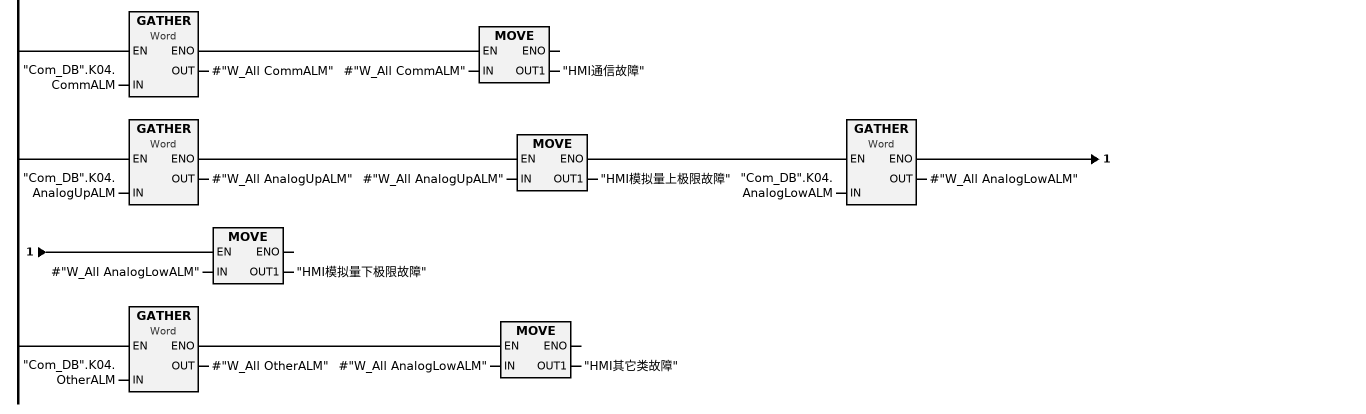
   RUNG wire#powerrail
      { S7_Templates := "[dest_type := Word, src_type := Bool]" } GATHER(IN := "Com_DB".K04.EMO, OUT => #"W_All EMO")
      Move(in := #"W_All EMO", out1 => "HMI总急停报警")
   END_RUNG
   RUNG wire#powerrail
      { S7_Templates := "[dest_type := Word, src_type := Bool]" } GATHER(IN := "Com_DB".K04.SLC, OUT => #"W_All SLC")
      Move(in := #"W_All SLC", out1 => "HMI总光栅报警")
   END_RUNG
   RUNG wire#powerrail
      { S7_Templates := "[dest_type := Word, src_type := Bool]" } GATHER(IN := "Com_DB".K04.DSW, OUT => #"W_All DSW")
      Move(in := #"W_All DSW", out1 => "HMI总安全门报警")
   END_RUNG
   RUNG wire#powerrail
      { S7_Templates := "[dest_type := Word, src_type := Bool]" } GATHER(IN := "Com_DB".K04.OtherSafe, OUT => #"W_All OtherSafe")
      Move(in := #"W_All OtherSafe", out1 => "HMI总其它安全报警")
   END_RUNG
   RUNG wire#powerrail
      { S7_Templates := "[dest_type := Word, src_type := Bool]" } GATHER(IN := "Com_DB".K04.AirALM, OUT => #"W_All AirALM")
      Move(in := #"W_All AirALM", out1 => "HMI总气压报警")
   END_RUNG
   RUNG wire#powerrail
      { S7_Templates := "[dest_type := Word, src_type := Bool, count_type := USInt]" } GATHER_BLK(IN := "Com_DB".K04.SensALM[1], COUNT_OUT := 6, OUT => #"W_All SensALM"[1])
      wire#w1
      Move(in := #"W_All SensALM"[1], out1 => "HMI传感器故障1")
   END_RUNG
   RUNG wire#w1
      Move(in := #"W_All SensALM"[2], out1 => "HMI传感器故障2")
   END_RUNG
   RUNG wire#w1
      Move(in := #"W_All SensALM"[3], out1 => "HMI传感器故障3")
   END_RUNG
   RUNG wire#w1
      Move(in := #"W_All SensALM"[4], out1 => "HMI传感器故障4")
   END_RUNG
   RUNG wire#w1
      Move(in := #"W_All SensALM"[5], out1 => "HMI传感器故障5")
   END_RUNG
   RUNG wire#w1
      Move(in := #"W_All SensALM"[6], out1 => "HMI传感器故障6")
   END_RUNG
   RUNG wire#powerrail
      { S7_Templates := "[dest_type := Word, src_type := Bool, count_type := USInt]" } GATHER_BLK(IN := "Com_DB".K04.MoveALM[1], COUNT_OUT := 3, OUT => #"W_All MoveALM"[1])
      wire#w2
      Move(in := #"W_All MoveALM"[1], out1 => "HMI动作异常1")
   END_RUNG
   RUNG wire#w2
      Move(in := #"W_All MoveALM"[2], out1 => "HMI动作异常2")
   END_RUNG
   RUNG wire#w2
      Move(in := #"W_All MoveALM"[3], out1 => "HMI动作异常3")
   END_RUNG
   RUNG wire#powerrail
      { S7_Templates := "[dest_type := Word, src_type := Bool, count_type := USInt]" } GATHER_BLK(IN := "Com_DB".K04.DrumALM[1], COUNT_OUT := 3, OUT => #"W_All DrumALM"[1])
      wire#w3
      Move(in := #"W_All DrumALM"[1], out1 => "HMI总滚筒故障1")
   END_RUNG
   RUNG wire#w3
      Move(in := #"W_All DrumALM"[2], out1 => "HMI总滚筒故障2")
   END_RUNG
   RUNG wire#w3
      Move(in := #"W_All DrumALM"[1], out1 => "HMI总滚筒故障3")
   END_RUNG
   RUNG wire#powerrail
      { S7_Templates := "[dest_type := Word, src_type := Bool, count_type := USInt]" } GATHER_BLK(IN := "Com_DB".K04.DrumTiOver[1], COUNT_OUT := 3, OUT => #"W_All DrumTiOver"[1])
      wire#w4
      Move(in := #"W_All DrumTiOver"[1], out1 => "HMI总滚筒超时1")
   END_RUNG
   RUNG wire#w4
      Move(in := #"W_All DrumTiOver"[2], out1 => "HMI总滚筒超时2")
   END_RUNG
   RUNG wire#w4
      Move(in := #"W_All DrumTiOver"[3], out1 => "HMI总滚筒超时3")
   END_RUNG
   RUNG wire#powerrail
      { S7_Templates := "[dest_type := Word, src_type := Bool]" } GATHER(IN := "Com_DB".K04.InvALM, OUT => #"W_All InvALM")
      Move(in := #"W_All InvALM", out1 => "HMI总变频器故障")
   END_RUNG
   RUNG wire#powerrail
      { S7_Templates := "[dest_type := Word, src_type := Bool]" } GATHER(IN := "Com_DB".K04.InvNoRun, OUT => #"W_All InvNoRun")
      Move(in := #"W_All InvNoRun", out1 => "HMI总变频器未运行故障")
   END_RUNG
   RUNG wire#powerrail
      { S7_Templates := "[dest_type := Word, src_type := Bool]" } GATHER(IN := "Com_DB".K04.InvOverload, OUT => #"W_All InvOverload")
      Move(in := #"W_All InvOverload", out1 => "HMI总变频器过载故障")
   END_RUNG
   RUNG wire#powerrail
      { S7_Templates := "[dest_type := Word, src_type := Bool]" } GATHER(IN := "Com_DB".K04.InvTiOver, OUT => #"W_All InvTiOver")
      Move(in := #"W_All InvTiOver", out1 => "HMI总变频器超时故障")
   END_RUNG
   RUNG wire#powerrail
      { S7_Templates := "[dest_type := Word, src_type := Bool, count_type := USInt]" } GATHER_BLK(IN := "Com_DB".K04.ValAdvTiOver[1], COUNT_OUT := 3, OUT => #"W_All ValAdvTiOver"[1])
      wire#w5
      { S7_Templates := "[dest_type := Word, src_type := Bool, count_type := USInt]" } GATHER_BLK(IN := "Com_DB".K04.ValRetTiOver[1], COUNT_OUT := 3, OUT => #"W_All ValRetTiOver"[1])
      wire#w6
      Move(in := #"W_All ValRetTiOver"[1], out1 => "HMI阀回动作超时1")
   END_RUNG
   RUNG wire#w6
      Move(in := #"W_All ValRetTiOver"[2], out1 => "HMI阀回动作超时2")
   END_RUNG
   RUNG wire#w6
      Move(in := #"W_All ValRetTiOver"[3], out1 => "HMI阀回动作超时3")
   END_RUNG
   RUNG wire#w5
      Move(in := #"W_All ValAdvTiOver"[1], out1 => "HMI阀出动作超时1")
   END_RUNG
   RUNG wire#w5
      Move(in := #"W_All ValAdvTiOver"[2], out1 => "HMI阀出动作超时2")
   END_RUNG
   RUNG wire#w5
      Move(in := #"W_All ValAdvTiOver"[3], out1 => "HMI阀出动作超时3")
   END_RUNG
   RUNG wire#powerrail
      { S7_Templates := "[dest_type := Word, src_type := Bool, count_type := USInt]" } GATHER_BLK(IN := "Com_DB".K04.ValSensALM[1], COUNT_OUT := 3, OUT => #"W_All ValSensALM"[1])
      wire#w7
      { S7_Templates := "[dest_type := Word, src_type := Bool, count_type := USInt]" } GATHER_BLK(IN := "Com_DB".K04.ValSenCroALM[1], COUNT_OUT := 3, OUT => #"W_All ValSenCroALM"[1])
      wire#w8
      Move(in := #"W_All ValSenCroALM"[1], out1 => "HMI阀传感器交叉ON故障1")
   END_RUNG
   RUNG wire#w8
      Move(in := #"W_All ValSenCroALM"[2], out1 => "HMI阀传感器交叉ON故障2")
   END_RUNG
   RUNG wire#w8
      Move(in := #"W_All ValSenCroALM"[3], out1 => "HMI阀传感器交叉ON故障3")
   END_RUNG
   RUNG wire#w7
      Move(in := #"W_All ValSensALM"[1], out1 => "HMI阀传感器全到位故障1")
   END_RUNG
   RUNG wire#w7
      Move(in := #"W_All ValSensALM"[2], out1 => "HMI阀传感器全到位故障2")
   END_RUNG
   RUNG wire#w7
      Move(in := #"W_All ValSensALM"[3], out1 => "HMI阀传感器全到位故障3")
   END_RUNG
   RUNG wire#powerrail
      { S7_Templates := "[dest_type := Word, src_type := Bool]" } GATHER(IN := "Com_DB".K04.AxisWarn, OUT => #"W_All AxisALM")
      Move(in := #"W_All AxisALM", out1 => "HMI伺服报警")
      { S7_Templates := "[dest_type := Word, src_type := Bool]" } GATHER(IN := "Com_DB".K04.AxisALM, OUT => #"W_All AxisERR")
      Move(in := #"W_All AxisERR", out1 => "HMI伺服故障")
   END_RUNG
   RUNG wire#powerrail
      { S7_Templates := "[dest_type := Word, src_type := Bool]" } GATHER(IN := "Com_DB".K04.AxisNoReady, OUT => #"W_All AxisReady")
      Move(in := #"W_All AxisReady", out1 => "HMI伺服未准备好")
      { S7_Templates := "[dest_type := Word, src_type := Bool]" } GATHER(IN := "Com_DB".K04.AxisHomeALM, OUT => #"W_All AxisHomeALM")
      Move(in := #"W_All AxisHomeALM", out1 => "HMI伺服未回零故障")
   END_RUNG
   RUNG wire#powerrail
      { S7_Templates := "[dest_type := Word, src_type := Bool]" } GATHER(IN := "Com_DB".K04.AxisNoRun, OUT => #"W_All AxisNoRun")
      Move(in := #"W_All AxisNoRun", out1 => "HMI伺服未运行故障")
   END_RUNG
   RUNG wire#powerrail
      { S7_Templates := "[dest_type := Word, src_type := Bool]" } GATHER(IN := "Com_DB".K04.AxisFLS, OUT => #"W_ALL AxisFLSALM")
      Move(in := #"W_ALL AxisFLSALM", out1 => "HM伺服正极限故障")
      { S7_Templates := "[dest_type := Word, src_type := Bool]" } GATHER(IN := "Com_DB".K04.AxisRLS, OUT => #"W_All AxisRLSALM")
      Move(in := #"W_All AxisRLSALM", out1 => "HMI伺服负极限故障")
   END_RUNG
   RUNG wire#powerrail
      { S7_Templates := "[dest_type := Word, src_type := Bool]" } GATHER(IN := "Com_DB".K04.RobotALM, OUT => #"W_All RobotALM")
      Move(in := #"W_All RobotALM", out1 => "HMI机器人故障")
   END_RUNG
   RUNG wire#powerrail
      { S7_Templates := "[dest_type := Word, src_type := Bool]" } GATHER(IN := "Com_DB".K04.CCDALM, OUT => #"W_All CCDALM")
      Move(in := #"W_All CCDALM", out1 => "HMI视觉故障")
   END_RUNG
   RUNG wire#powerrail
      { S7_Templates := "[dest_type := Word, src_type := Bool]" } GATHER(IN := "Com_DB".K04.CommALM, OUT => #"W_All CommALM")
      Move(in := #"W_All CommALM", out1 => "HMI通信故障")
   END_RUNG
   RUNG wire#powerrail
      { S7_Templates := "[dest_type := Word, src_type := Bool]" } GATHER(IN := "Com_DB".K04.AnalogUpALM, OUT => #"W_All AnalogUpALM")
      Move(in := #"W_All AnalogUpALM", out1 => "HMI模拟量上极限故障")
      { S7_Templates := "[dest_type := Word, src_type := Bool]" } GATHER(IN := "Com_DB".K04.AnalogLowALM, OUT => #"W_All AnalogLowALM")
      Move(in := #"W_All AnalogLowALM", out1 => "HMI模拟量下极限故障")
   END_RUNG
   RUNG wire#powerrail
      { S7_Templates := "[dest_type := Word, src_type := Bool]" } GATHER(IN := "Com_DB".K04.OtherALM, OUT => #"W_All OtherALM")
      Move(in := #"W_All AnalogLowALM", out1 => "HMI其它类故障")
   END_RUNG
   // the same network as SCL:
   GATHER(IN := "Com_DB".K04.EMO, OUT => #"W_All EMO", ENO => #_w1);
   IF #_w1 THEN "HMI总急停报警" := #"W_All EMO"; END_IF;
   GATHER(IN := "Com_DB".K04.SLC, OUT => #"W_All SLC", ENO => #_w2);
   IF #_w2 THEN "HMI总光栅报警" := #"W_All SLC"; END_IF;
   GATHER(IN := "Com_DB".K04.DSW, OUT => #"W_All DSW", ENO => #_w3);
   IF #_w3 THEN "HMI总安全门报警" := #"W_All DSW"; END_IF;
   GATHER(IN := "Com_DB".K04.OtherSafe, OUT => #"W_All OtherSafe", ENO => #_w4);
   IF #_w4 THEN "HMI总其它安全报警" := #"W_All OtherSafe"; END_IF;
   GATHER(IN := "Com_DB".K04.AirALM, OUT => #"W_All AirALM", ENO => #_w5);
   IF #_w5 THEN "HMI总气压报警" := #"W_All AirALM"; END_IF;
   GATHER_BLK(IN := "Com_DB".K04.SensALM[1], COUNT_OUT := 6, OUT => #"W_All SensALM"[1], ENO => #_w6);
   IF #_w6 THEN
       "HMI传感器故障1" := #"W_All SensALM"[1];
       "HMI传感器故障2" := #"W_All SensALM"[2];
       "HMI传感器故障3" := #"W_All SensALM"[3];
       "HMI传感器故障4" := #"W_All SensALM"[4];
       "HMI传感器故障5" := #"W_All SensALM"[5];
       "HMI传感器故障6" := #"W_All SensALM"[6];
   END_IF;
   GATHER_BLK(IN := "Com_DB".K04.MoveALM[1], COUNT_OUT := 3, OUT => #"W_All MoveALM"[1], ENO => #_w7);
   IF #_w7 THEN
       "HMI动作异常1" := #"W_All MoveALM"[1];
       "HMI动作异常2" := #"W_All MoveALM"[2];
       "HMI动作异常3" := #"W_All MoveALM"[3];
   END_IF;
   GATHER_BLK(IN := "Com_DB".K04.DrumALM[1], COUNT_OUT := 3, OUT => #"W_All DrumALM"[1], ENO => #_w8);
   IF #_w8 THEN
       "HMI总滚筒故障1" := #"W_All DrumALM"[1];
       "HMI总滚筒故障2" := #"W_All DrumALM"[2];
       "HMI总滚筒故障3" := #"W_All DrumALM"[1];
   END_IF;
   GATHER_BLK(IN := "Com_DB".K04.DrumTiOver[1], COUNT_OUT := 3, OUT => #"W_All DrumTiOver"[1], ENO => #_w9);
   IF #_w9 THEN
       "HMI总滚筒超时1" := #"W_All DrumTiOver"[1];
       "HMI总滚筒超时2" := #"W_All DrumTiOver"[2];
       "HMI总滚筒超时3" := #"W_All DrumTiOver"[3];
   END_IF;
   GATHER(IN := "Com_DB".K04.InvALM, OUT => #"W_All InvALM", ENO => #_w10);
   IF #_w10 THEN "HMI总变频器故障" := #"W_All InvALM"; END_IF;
   GATHER(IN := "Com_DB".K04.InvNoRun, OUT => #"W_All InvNoRun", ENO => #_w11);
   IF #_w11 THEN "HMI总变频器未运行故障" := #"W_All InvNoRun"; END_IF;
   GATHER(IN := "Com_DB".K04.InvOverload, OUT => #"W_All InvOverload", ENO => #_w12);
   IF #_w12 THEN "HMI总变频器过载故障" := #"W_All InvOverload"; END_IF;
   GATHER(IN := "Com_DB".K04.InvTiOver, OUT => #"W_All InvTiOver", ENO => #_w13);
   IF #_w13 THEN "HMI总变频器超时故障" := #"W_All InvTiOver"; END_IF;
   GATHER_BLK(IN := "Com_DB".K04.ValAdvTiOver[1], COUNT_OUT := 3, OUT => #"W_All ValAdvTiOver"[1], ENO => #_w14);
   GATHER_BLK(EN := #_w14,
              IN := "Com_DB".K04.ValRetTiOver[1],
              COUNT_OUT := 3,
              OUT => #"W_All ValRetTiOver"[1],
              ENO => #_w15);
   IF #_w15 THEN
       "HMI阀回动作超时1" := #"W_All ValRetTiOver"[1];
       "HMI阀回动作超时2" := #"W_All ValRetTiOver"[2];
       "HMI阀回动作超时3" := #"W_All ValRetTiOver"[3];
   END_IF;
   IF #_w14 THEN
       "HMI阀出动作超时1" := #"W_All ValAdvTiOver"[1];
       "HMI阀出动作超时2" := #"W_All ValAdvTiOver"[2];
       "HMI阀出动作超时3" := #"W_All ValAdvTiOver"[3];
   END_IF;
   GATHER_BLK(IN := "Com_DB".K04.ValSensALM[1], COUNT_OUT := 3, OUT => #"W_All ValSensALM"[1], ENO => #_w16);
   GATHER_BLK(EN := #_w16,
              IN := "Com_DB".K04.ValSenCroALM[1],
              COUNT_OUT := 3,
              OUT => #"W_All ValSenCroALM"[1],
              ENO => #_w17);
   IF #_w17 THEN
       "HMI阀传感器交叉ON故障1" := #"W_All ValSenCroALM"[1];
       "HMI阀传感器交叉ON故障2" := #"W_All ValSenCroALM"[2];
       "HMI阀传感器交叉ON故障3" := #"W_All ValSenCroALM"[3];
   END_IF;
   IF #_w16 THEN
       "HMI阀传感器全到位故障1" := #"W_All ValSensALM"[1];
       "HMI阀传感器全到位故障2" := #"W_All ValSensALM"[2];
       "HMI阀传感器全到位故障3" := #"W_All ValSensALM"[3];
   END_IF;
   GATHER(IN := "Com_DB".K04.AxisWarn, OUT => #"W_All AxisALM", ENO => #_w18);
   IF #_w18 THEN "HMI伺服报警" := #"W_All AxisALM"; END_IF;
   GATHER(EN := #_w18, IN := "Com_DB".K04.AxisALM, OUT => #"W_All AxisERR", ENO => #_w19);
   IF #_w19 THEN "HMI伺服故障" := #"W_All AxisERR"; END_IF;
   GATHER(IN := "Com_DB".K04.AxisNoReady, OUT => #"W_All AxisReady", ENO => #_w20);
   IF #_w20 THEN "HMI伺服未准备好" := #"W_All AxisReady"; END_IF;
   GATHER(EN := #_w20, IN := "Com_DB".K04.AxisHomeALM, OUT => #"W_All AxisHomeALM", ENO => #_w21);
   IF #_w21 THEN "HMI伺服未回零故障" := #"W_All AxisHomeALM"; END_IF;
   GATHER(IN := "Com_DB".K04.AxisNoRun, OUT => #"W_All AxisNoRun", ENO => #_w22);
   IF #_w22 THEN "HMI伺服未运行故障" := #"W_All AxisNoRun"; END_IF;
   GATHER(IN := "Com_DB".K04.AxisFLS, OUT => #"W_ALL AxisFLSALM", ENO => #_w23);
   IF #_w23 THEN "HM伺服正极限故障" := #"W_ALL AxisFLSALM"; END_IF;
   GATHER(EN := #_w23, IN := "Com_DB".K04.AxisRLS, OUT => #"W_All AxisRLSALM", ENO => #_w24);
   IF #_w24 THEN "HMI伺服负极限故障" := #"W_All AxisRLSALM"; END_IF;
   GATHER(IN := "Com_DB".K04.RobotALM, OUT => #"W_All RobotALM", ENO => #_w25);
   IF #_w25 THEN "HMI机器人故障" := #"W_All RobotALM"; END_IF;
   GATHER(IN := "Com_DB".K04.CCDALM, OUT => #"W_All CCDALM", ENO => #_w26);
   IF #_w26 THEN "HMI视觉故障" := #"W_All CCDALM"; END_IF;
   GATHER(IN := "Com_DB".K04.CommALM, OUT => #"W_All CommALM", ENO => #_w27);
   IF #_w27 THEN "HMI通信故障" := #"W_All CommALM"; END_IF;
   GATHER(IN := "Com_DB".K04.AnalogUpALM, OUT => #"W_All AnalogUpALM", ENO => #_w28);
   IF #_w28 THEN "HMI模拟量上极限故障" := #"W_All AnalogUpALM"; END_IF;
   GATHER(EN := #_w28, IN := "Com_DB".K04.AnalogLowALM, OUT => #"W_All AnalogLowALM", ENO => #_w29);
   IF #_w29 THEN "HMI模拟量下极限故障" := #"W_All AnalogLowALM"; END_IF;
   GATHER(IN := "Com_DB".K04.OtherALM, OUT => #"W_All OtherALM", ENO => #_w30);
   IF #_w30 THEN "HMI其它类故障" := #"W_All AnalogLowALM"; END_IF;
END_REGION

REGION Network 18: 安全类
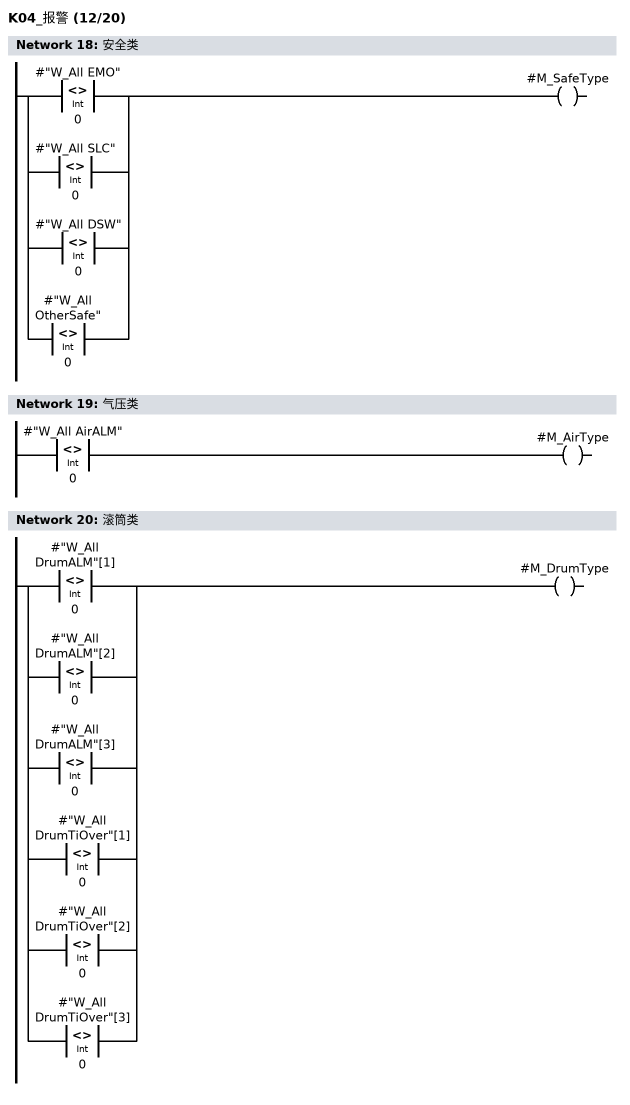
   RUNG wire#powerrail
      { S7_Templates := "SrcType := Int" } NE_Contact(in1 := #"W_All EMO", in2 := 0)
      wire#w1
      Coil( #M_SafeType )
   END_RUNG
   RUNG wire#powerrail
      { S7_Templates := "SrcType := Int" } NE_Contact(in1 := #"W_All SLC", in2 := 0)
   END_RUNG wire#w1
   RUNG wire#powerrail
      { S7_Templates := "SrcType := Int" } NE_Contact(in1 := #"W_All DSW", in2 := 0)
   END_RUNG wire#w1
   RUNG wire#powerrail
      { S7_Templates := "SrcType := Int" } NE_Contact(in1 := #"W_All OtherSafe", in2 := 0)
   END_RUNG wire#w1
   // the same network as SCL:
   #M_SafeType := (#"W_All EMO" <> 0) OR (#"W_All SLC" <> 0) OR (#"W_All DSW" <> 0) OR (#"W_All OtherSafe" <> 0);
END_REGION

REGION Network 19: 气压类
   RUNG wire#powerrail
      { S7_Templates := "SrcType := Int" } NE_Contact(in1 := #"W_All AirALM", in2 := 0)
      Coil( #M_AirType )
   END_RUNG
   // the same network as SCL:
   #M_AirType := #"W_All AirALM" <> 0;
END_REGION

REGION Network 20: 滚筒类
   RUNG wire#powerrail
      { S7_Templates := "SrcType := Int" } NE_Contact(in1 := #"W_All DrumALM"[1], in2 := 0)
      wire#w1
      Coil( #M_DrumType )
   END_RUNG
   RUNG wire#powerrail
      { S7_Templates := "SrcType := Int" } NE_Contact(in1 := #"W_All DrumALM"[2], in2 := 0)
   END_RUNG wire#w1
   RUNG wire#powerrail
      { S7_Templates := "SrcType := Int" } NE_Contact(in1 := #"W_All DrumALM"[3], in2 := 0)
   END_RUNG wire#w1
   RUNG wire#powerrail
      { S7_Templates := "SrcType := Int" } NE_Contact(in1 := #"W_All DrumTiOver"[1], in2 := 0)
   END_RUNG wire#w1
   RUNG wire#powerrail
      { S7_Templates := "SrcType := Int" } NE_Contact(in1 := #"W_All DrumTiOver"[2], in2 := 0)
   END_RUNG wire#w1
   RUNG wire#powerrail
      { S7_Templates := "SrcType := Int" } NE_Contact(in1 := #"W_All DrumTiOver"[3], in2 := 0)
   END_RUNG wire#w1
   // the same network as SCL:
   #M_DrumType := (#"W_All DrumALM"[1] <> 0) OR (#"W_All DrumALM"[2] <> 0) OR (#"W_All DrumALM"[3] <> 0) OR (#"W_All DrumTiOver"[1] <> 0) OR (#"W_All DrumTiOver"[2] <> 0) OR (#"W_All DrumTiOver"[3] <> 0);
END_REGION

REGION Network 21: 变频器类
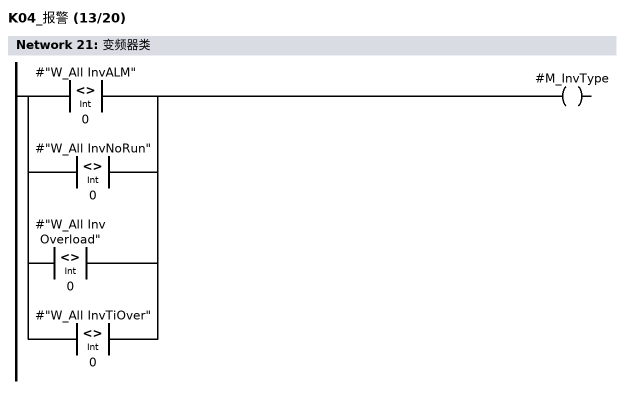
   RUNG wire#powerrail
      { S7_Templates := "SrcType := Int" } NE_Contact(in1 := #"W_All InvALM", in2 := 0)
      wire#w1
      Coil( #M_InvType )
   END_RUNG
   RUNG wire#powerrail
      { S7_Templates := "SrcType := Int" } NE_Contact(in1 := #"W_All InvNoRun", in2 := 0)
   END_RUNG wire#w1
   RUNG wire#powerrail
      { S7_Templates := "SrcType := Int" } NE_Contact(in1 := #"W_All InvOverload", in2 := 0)
   END_RUNG wire#w1
   RUNG wire#powerrail
      { S7_Templates := "SrcType := Int" } NE_Contact(in1 := #"W_All InvTiOver", in2 := 0)
   END_RUNG wire#w1
   // the same network as SCL:
   #M_InvType := (#"W_All InvALM" <> 0) OR (#"W_All InvNoRun" <> 0) OR (#"W_All InvOverload" <> 0) OR (#"W_All InvTiOver" <> 0);
END_REGION

REGION Network 22: 阀类型故障
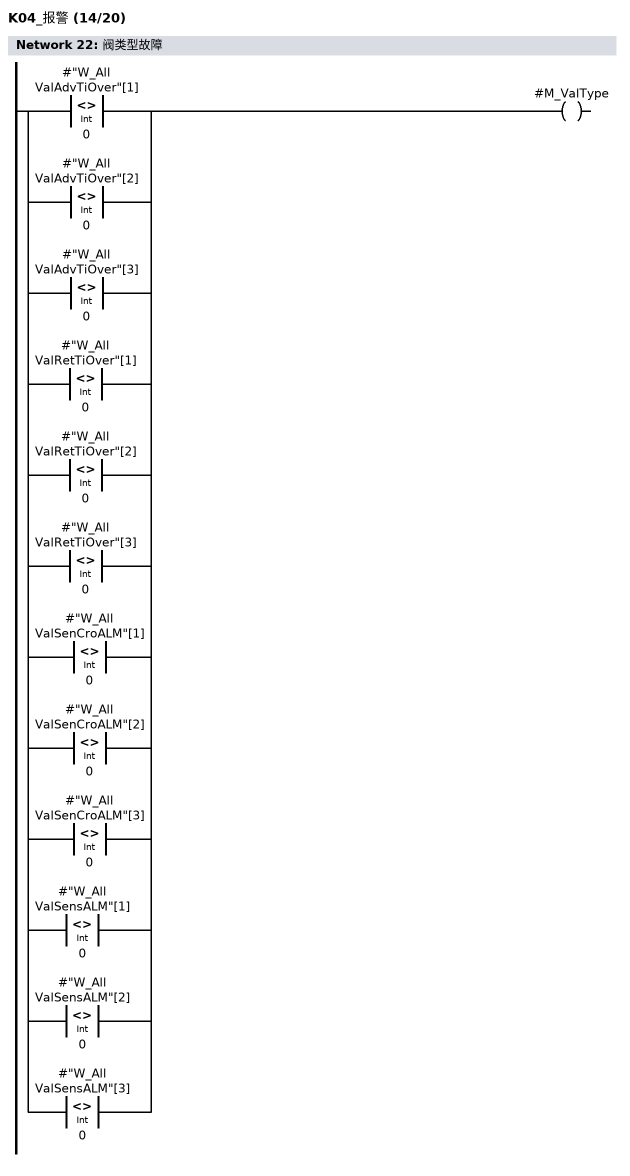
   RUNG wire#powerrail
      { S7_Templates := "SrcType := Int" } NE_Contact(in1 := #"W_All ValAdvTiOver"[1], in2 := 0)
      wire#w1
      Coil( #M_ValType )
   END_RUNG
   RUNG wire#powerrail
      { S7_Templates := "SrcType := Int" } NE_Contact(in1 := #"W_All ValAdvTiOver"[2], in2 := 0)
   END_RUNG wire#w1
   RUNG wire#powerrail
      { S7_Templates := "SrcType := Int" } NE_Contact(in1 := #"W_All ValAdvTiOver"[3], in2 := 0)
   END_RUNG wire#w1
   RUNG wire#powerrail
      { S7_Templates := "SrcType := Int" } NE_Contact(in1 := #"W_All ValRetTiOver"[1], in2 := 0)
   END_RUNG wire#w1
   RUNG wire#powerrail
      { S7_Templates := "SrcType := Int" } NE_Contact(in1 := #"W_All ValRetTiOver"[2], in2 := 0)
   END_RUNG wire#w1
   RUNG wire#powerrail
      { S7_Templates := "SrcType := Int" } NE_Contact(in1 := #"W_All ValRetTiOver"[3], in2 := 0)
   END_RUNG wire#w1
   RUNG wire#powerrail
      { S7_Templates := "SrcType := Int" } NE_Contact(in1 := #"W_All ValSenCroALM"[1], in2 := 0)
   END_RUNG wire#w1
   RUNG wire#powerrail
      { S7_Templates := "SrcType := Int" } NE_Contact(in1 := #"W_All ValSenCroALM"[2], in2 := 0)
   END_RUNG wire#w1
   RUNG wire#powerrail
      { S7_Templates := "SrcType := Int" } NE_Contact(in1 := #"W_All ValSenCroALM"[3], in2 := 0)
   END_RUNG wire#w1
   RUNG wire#powerrail
      { S7_Templates := "SrcType := Int" } NE_Contact(in1 := #"W_All ValSensALM"[1], in2 := 0)
   END_RUNG wire#w1
   RUNG wire#powerrail
      { S7_Templates := "SrcType := Int" } NE_Contact(in1 := #"W_All ValSensALM"[2], in2 := 0)
   END_RUNG wire#w1
   RUNG wire#powerrail
      { S7_Templates := "SrcType := Int" } NE_Contact(in1 := #"W_All ValSensALM"[3], in2 := 0)
   END_RUNG wire#w1
   // the same network as SCL:
   #M_ValType := (#"W_All ValAdvTiOver"[1] <> 0) OR (#"W_All ValAdvTiOver"[2] <> 0) OR (#"W_All ValAdvTiOver"[3] <> 0) OR (#"W_All ValRetTiOver"[1] <> 0) OR (#"W_All ValRetTiOver"[2] <> 0) OR (#"W_All ValRetTiOver"[3] <> 0) OR (#"W_All ValSenCroALM"[1] <> 0) OR (#"W_All ValSenCroALM"[2] <> 0) OR (#"W_All ValSenCroALM"[3] <> 0) OR (#"W_All ValSensALM"[1] <> 0) OR (#"W_All ValSensALM"[2] <> 0) OR (#"W_All ValSensALM"[3] <> 0);
END_REGION

REGION Network 23: 伺服类别
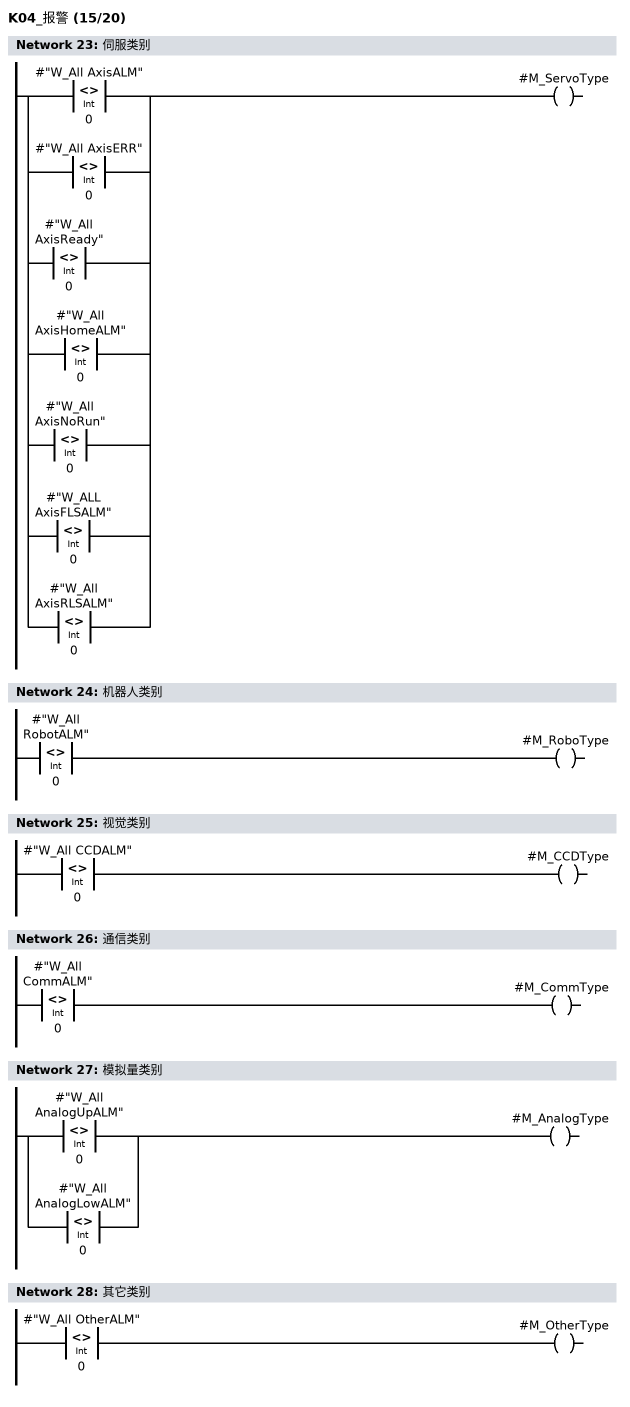
   RUNG wire#powerrail
      { S7_Templates := "SrcType := Int" } NE_Contact(in1 := #"W_All AxisALM", in2 := 0)
      wire#w1
      Coil( #M_ServoType )
   END_RUNG
   RUNG wire#powerrail
      { S7_Templates := "SrcType := Int" } NE_Contact(in1 := #"W_All AxisERR", in2 := 0)
   END_RUNG wire#w1
   RUNG wire#powerrail
      { S7_Templates := "SrcType := Int" } NE_Contact(in1 := #"W_All AxisReady", in2 := 0)
   END_RUNG wire#w1
   RUNG wire#powerrail
      { S7_Templates := "SrcType := Int" } NE_Contact(in1 := #"W_All AxisHomeALM", in2 := 0)
   END_RUNG wire#w1
   RUNG wire#powerrail
      { S7_Templates := "SrcType := Int" } NE_Contact(in1 := #"W_All AxisNoRun", in2 := 0)
   END_RUNG wire#w1
   RUNG wire#powerrail
      { S7_Templates := "SrcType := Int" } NE_Contact(in1 := #"W_ALL AxisFLSALM", in2 := 0)
   END_RUNG wire#w1
   RUNG wire#powerrail
      { S7_Templates := "SrcType := Int" } NE_Contact(in1 := #"W_All AxisRLSALM", in2 := 0)
   END_RUNG wire#w1
   // the same network as SCL:
   #M_ServoType := (#"W_All AxisALM" <> 0) OR (#"W_All AxisERR" <> 0) OR (#"W_All AxisReady" <> 0) OR (#"W_All AxisHomeALM" <> 0) OR (#"W_All AxisNoRun" <> 0) OR (#"W_ALL AxisFLSALM" <> 0) OR (#"W_All AxisRLSALM" <> 0);
END_REGION

REGION Network 24: 机器人类别
   RUNG wire#powerrail
      { S7_Templates := "SrcType := Int" } NE_Contact(in1 := #"W_All RobotALM", in2 := 0)
      Coil( #M_RoboType )
   END_RUNG
   // the same network as SCL:
   #M_RoboType := #"W_All RobotALM" <> 0;
END_REGION

REGION Network 25: 视觉类别
   RUNG wire#powerrail
      { S7_Templates := "SrcType := Int" } NE_Contact(in1 := #"W_All CCDALM", in2 := 0)
      Coil( #M_CCDType )
   END_RUNG
   // the same network as SCL:
   #M_CCDType := #"W_All CCDALM" <> 0;
END_REGION

REGION Network 26: 通信类别
   RUNG wire#powerrail
      { S7_Templates := "SrcType := Int" } NE_Contact(in1 := #"W_All CommALM", in2 := 0)
      Coil( #M_CommType )
   END_RUNG
   // the same network as SCL:
   #M_CommType := #"W_All CommALM" <> 0;
END_REGION

REGION Network 27: 模拟量类别
   RUNG wire#powerrail
      { S7_Templates := "SrcType := Int" } NE_Contact(in1 := #"W_All AnalogUpALM", in2 := 0)
      wire#w1
      Coil( #M_AnalogType )
   END_RUNG
   RUNG wire#powerrail
      { S7_Templates := "SrcType := Int" } NE_Contact(in1 := #"W_All AnalogLowALM", in2 := 0)
   END_RUNG wire#w1
   // the same network as SCL:
   #M_AnalogType := (#"W_All AnalogUpALM" <> 0) OR (#"W_All AnalogLowALM" <> 0);
END_REGION

REGION Network 28: 其它类别
   RUNG wire#powerrail
      { S7_Templates := "SrcType := Int" } NE_Contact(in1 := #"W_All OtherALM", in2 := 0)
      Coil( #M_OtherType )
   END_RUNG
   // the same network as SCL:
   #M_OtherType := #"W_All OtherALM" <> 0;
END_REGION

REGION Network 29: 传感器故障类
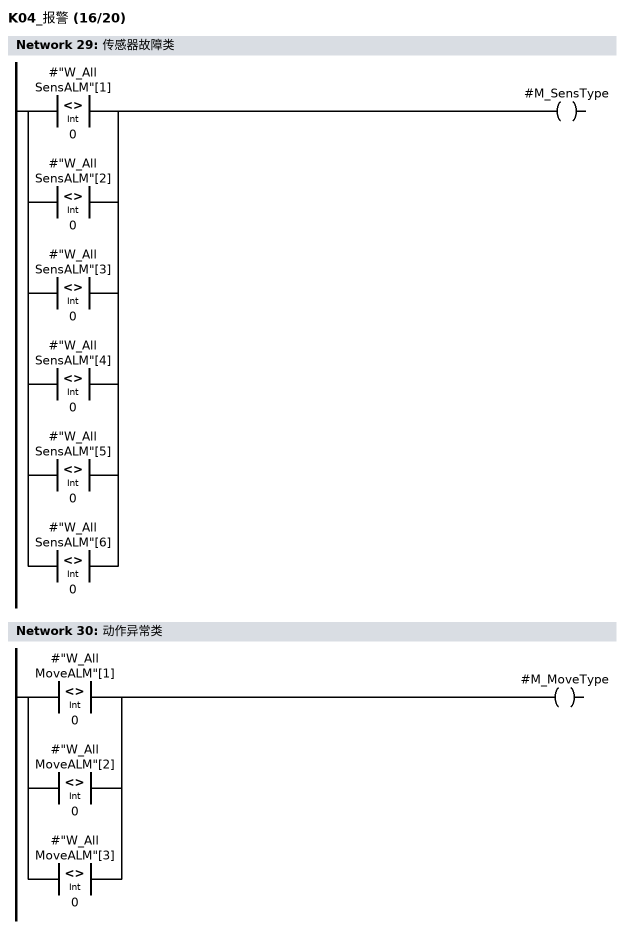
   RUNG wire#powerrail
      { S7_Templates := "SrcType := Int" } NE_Contact(in1 := #"W_All SensALM"[1], in2 := 0)
      wire#w1
      Coil( #M_SensType )
   END_RUNG
   RUNG wire#powerrail
      { S7_Templates := "SrcType := Int" } NE_Contact(in1 := #"W_All SensALM"[2], in2 := 0)
   END_RUNG wire#w1
   RUNG wire#powerrail
      { S7_Templates := "SrcType := Int" } NE_Contact(in1 := #"W_All SensALM"[3], in2 := 0)
   END_RUNG wire#w1
   RUNG wire#powerrail
      { S7_Templates := "SrcType := Int" } NE_Contact(in1 := #"W_All SensALM"[4], in2 := 0)
   END_RUNG wire#w1
   RUNG wire#powerrail
      { S7_Templates := "SrcType := Int" } NE_Contact(in1 := #"W_All SensALM"[5], in2 := 0)
   END_RUNG wire#w1
   RUNG wire#powerrail
      { S7_Templates := "SrcType := Int" } NE_Contact(in1 := #"W_All SensALM"[6], in2 := 0)
   END_RUNG wire#w1
   // the same network as SCL:
   #M_SensType := (#"W_All SensALM"[1] <> 0) OR (#"W_All SensALM"[2] <> 0) OR (#"W_All SensALM"[3] <> 0) OR (#"W_All SensALM"[4] <> 0) OR (#"W_All SensALM"[5] <> 0) OR (#"W_All SensALM"[6] <> 0);
END_REGION

REGION Network 30: 动作异常类
   RUNG wire#powerrail
      { S7_Templates := "SrcType := Int" } NE_Contact(in1 := #"W_All MoveALM"[1], in2 := 0)
      wire#w1
      Coil( #M_MoveType )
   END_RUNG
   RUNG wire#powerrail
      { S7_Templates := "SrcType := Int" } NE_Contact(in1 := #"W_All MoveALM"[2], in2 := 0)
   END_RUNG wire#w1
   RUNG wire#powerrail
      { S7_Templates := "SrcType := Int" } NE_Contact(in1 := #"W_All MoveALM"[3], in2 := 0)
   END_RUNG wire#w1
   // the same network as SCL:
   #M_MoveType := (#"W_All MoveALM"[1] <> 0) OR (#"W_All MoveALM"[2] <> 0) OR (#"W_All MoveALM"[3] <> 0);
END_REGION

REGION Network 31: 故障汇总
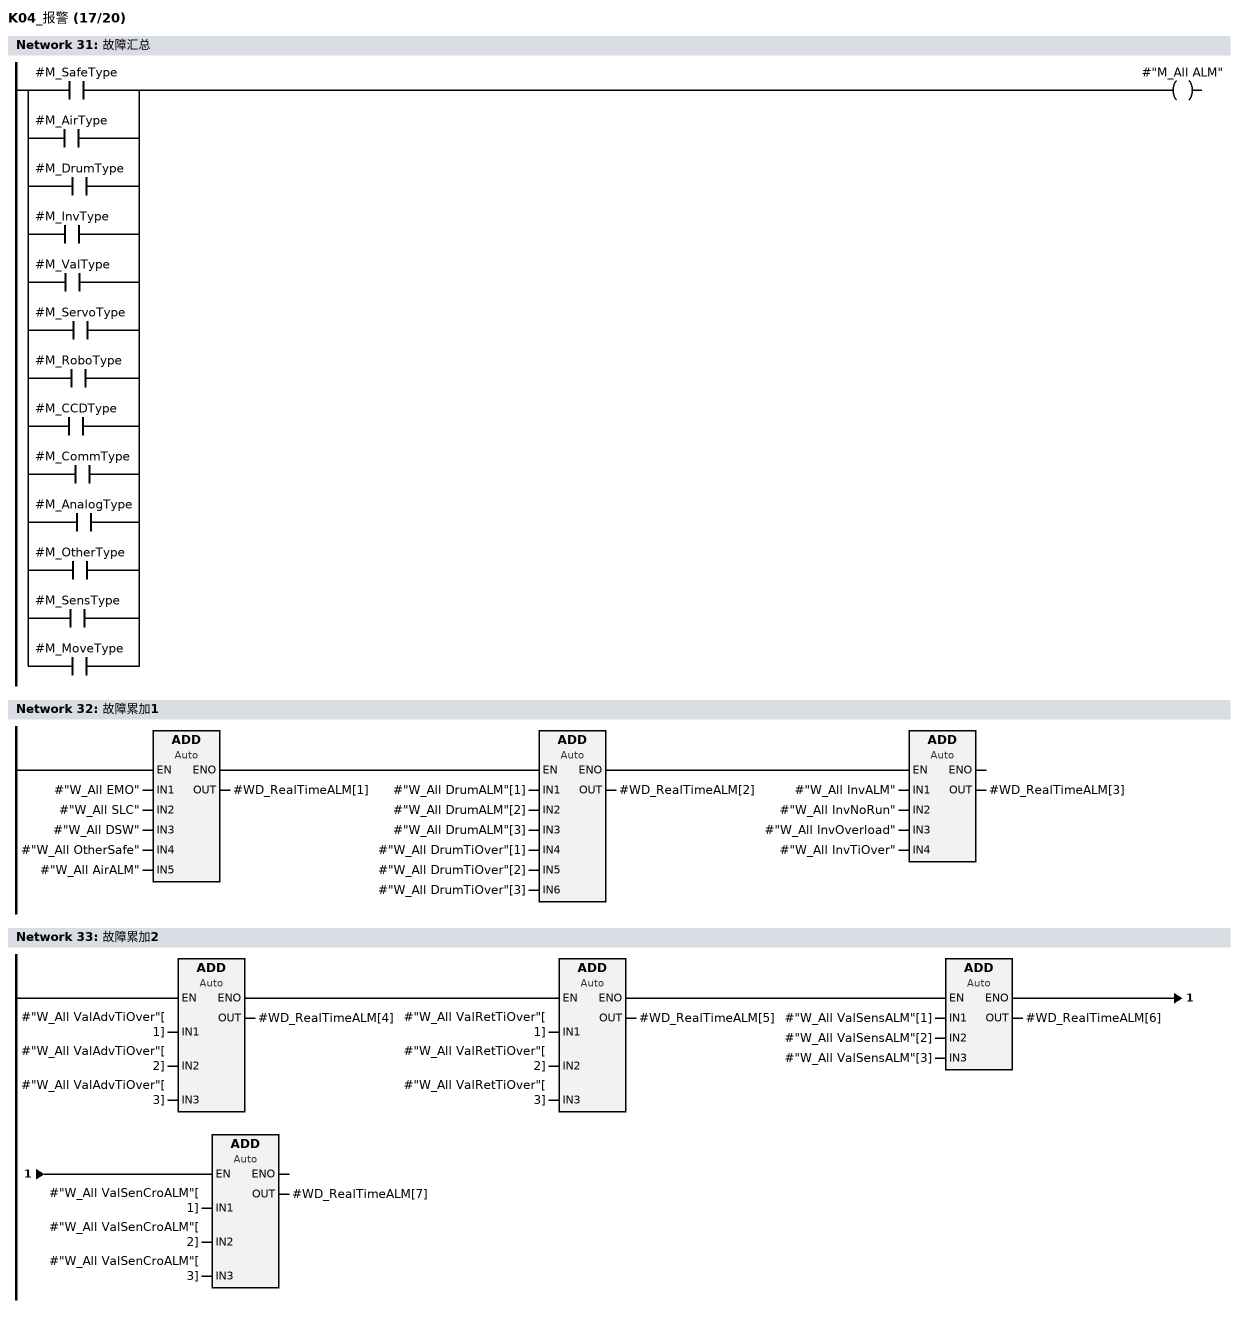
   RUNG wire#powerrail
      Contact( #M_SafeType )
      wire#w1
      Coil( #"M_All ALM" )
   END_RUNG
   RUNG wire#powerrail
      Contact( #M_AirType )
   END_RUNG wire#w1
   RUNG wire#powerrail
      Contact( #M_DrumType )
   END_RUNG wire#w1
   RUNG wire#powerrail
      Contact( #M_InvType )
   END_RUNG wire#w1
   RUNG wire#powerrail
      Contact( #M_ValType )
   END_RUNG wire#w1
   RUNG wire#powerrail
      Contact( #M_ServoType )
   END_RUNG wire#w1
   RUNG wire#powerrail
      Contact( #M_RoboType )
   END_RUNG wire#w1
   RUNG wire#powerrail
      Contact( #M_CCDType )
   END_RUNG wire#w1
   RUNG wire#powerrail
      Contact( #M_CommType )
   END_RUNG wire#w1
   RUNG wire#powerrail
      Contact( #M_AnalogType )
   END_RUNG wire#w1
   RUNG wire#powerrail
      Contact( #M_OtherType )
   END_RUNG wire#w1
   RUNG wire#powerrail
      Contact( #M_SensType )
   END_RUNG wire#w1
   RUNG wire#powerrail
      Contact( #M_MoveType )
   END_RUNG wire#w1
   // the same network as SCL:
   #"M_All ALM" := #M_SafeType OR #M_AirType OR #M_DrumType OR #M_InvType OR #M_ValType OR #M_ServoType OR #M_RoboType OR #M_CCDType OR #M_CommType OR #M_AnalogType OR #M_OtherType OR #M_SensType OR #M_MoveType;
END_REGION

REGION Network 32: 故障累加1
   RUNG wire#powerrail
      Add(in1 := #"W_All EMO", in2 := #"W_All SLC", in3 := #"W_All DSW", in4 := #"W_All OtherSafe", in5 := #"W_All AirALM", out => #WD_RealTimeALM[1])
      Add(in1 := #"W_All DrumALM"[1], in2 := #"W_All DrumALM"[2], in3 := #"W_All DrumALM"[3], in4 := #"W_All DrumTiOver"[1], in5 := #"W_All DrumTiOver"[2], in6 := #"W_All DrumTiOver"[3], out => #WD_RealTimeALM[2])
      Add(in1 := #"W_All InvALM", in2 := #"W_All InvNoRun", in3 := #"W_All InvOverload", in4 := #"W_All InvTiOver", out => #WD_RealTimeALM[3])
   END_RUNG
   // the same network as SCL:
   #WD_RealTimeALM[1] := #"W_All EMO" + #"W_All SLC" + #"W_All DSW" + #"W_All OtherSafe" + #"W_All AirALM";
   #WD_RealTimeALM[2] := #"W_All DrumALM"[1] + #"W_All DrumALM"[2] + #"W_All DrumALM"[3] + #"W_All DrumTiOver"[1] + #"W_All DrumTiOver"[2] + #"W_All DrumTiOver"[3];
   #WD_RealTimeALM[3] := #"W_All InvALM" + #"W_All InvNoRun" + #"W_All InvOverload" + #"W_All InvTiOver";
END_REGION

REGION Network 33: 故障累加2
   RUNG wire#powerrail
      Add(in1 := #"W_All ValAdvTiOver"[1], in2 := #"W_All ValAdvTiOver"[2], in3 := #"W_All ValAdvTiOver"[3], out => #WD_RealTimeALM[4])
      Add(in1 := #"W_All ValRetTiOver"[1], in2 := #"W_All ValRetTiOver"[2], in3 := #"W_All ValRetTiOver"[3], out => #WD_RealTimeALM[5])
      Add(in1 := #"W_All ValSensALM"[1], in2 := #"W_All ValSensALM"[2], in3 := #"W_All ValSensALM"[3], out => #WD_RealTimeALM[6])
      Add(in1 := #"W_All ValSenCroALM"[1], in2 := #"W_All ValSenCroALM"[2], in3 := #"W_All ValSenCroALM"[3], out => #WD_RealTimeALM[7])
   END_RUNG
   // the same network as SCL:
   #WD_RealTimeALM[4] := #"W_All ValAdvTiOver"[1] + #"W_All ValAdvTiOver"[2] + #"W_All ValAdvTiOver"[3];
   #WD_RealTimeALM[5] := #"W_All ValRetTiOver"[1] + #"W_All ValRetTiOver"[2] + #"W_All ValRetTiOver"[3];
   #WD_RealTimeALM[6] := #"W_All ValSensALM"[1] + #"W_All ValSensALM"[2] + #"W_All ValSensALM"[3];
   #WD_RealTimeALM[7] := #"W_All ValSenCroALM"[1] + #"W_All ValSenCroALM"[2] + #"W_All ValSenCroALM"[3];
END_REGION

REGION Network 34: 故障累加3
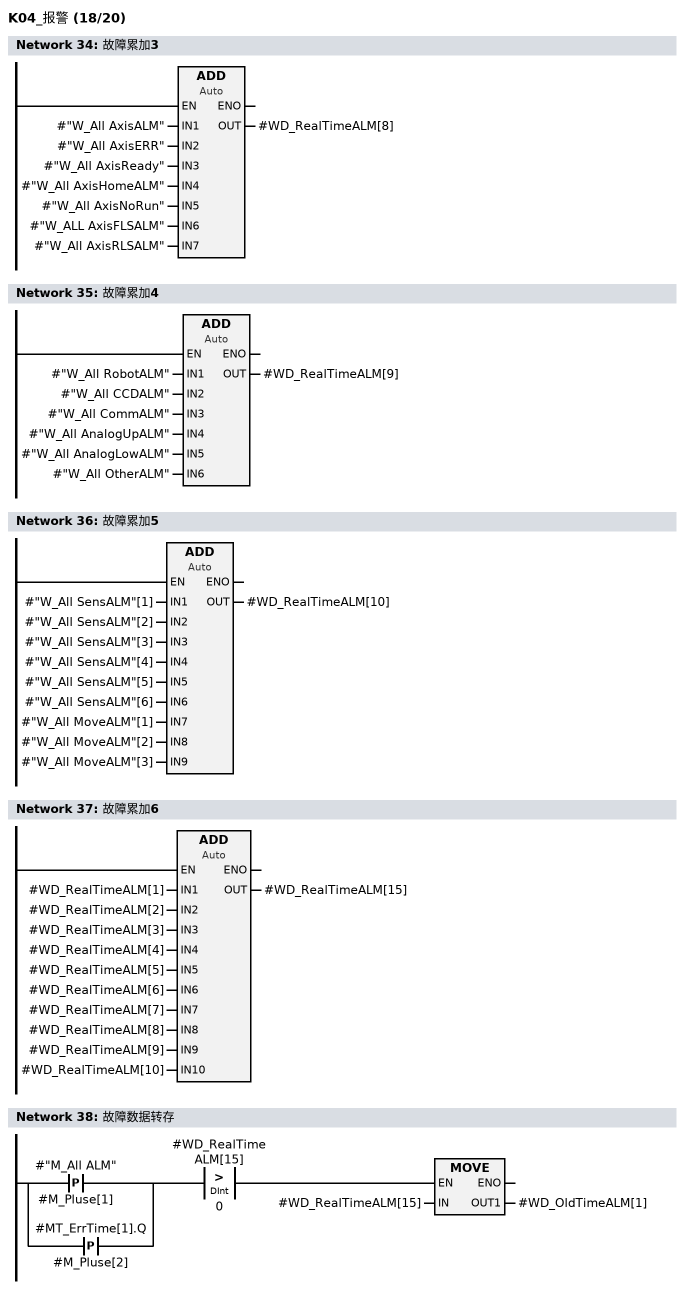
   RUNG wire#powerrail
      Add(in1 := #"W_All AxisALM", in2 := #"W_All AxisERR", in3 := #"W_All AxisReady", in4 := #"W_All AxisHomeALM", in5 := #"W_All AxisNoRun", in6 := #"W_ALL AxisFLSALM", in7 := #"W_All AxisRLSALM", out => #WD_RealTimeALM[8])
   END_RUNG
   // the same network as SCL:
   #WD_RealTimeALM[8] := #"W_All AxisALM" + #"W_All AxisERR" + #"W_All AxisReady" + #"W_All AxisHomeALM" + #"W_All AxisNoRun" + #"W_ALL AxisFLSALM" + #"W_All AxisRLSALM";
END_REGION

REGION Network 35: 故障累加4
   RUNG wire#powerrail
      Add(in1 := #"W_All RobotALM", in2 := #"W_All CCDALM", in3 := #"W_All CommALM", in4 := #"W_All AnalogUpALM", in5 := #"W_All AnalogLowALM", in6 := #"W_All OtherALM", out => #WD_RealTimeALM[9])
   END_RUNG
   // the same network as SCL:
   #WD_RealTimeALM[9] := #"W_All RobotALM" + #"W_All CCDALM" + #"W_All CommALM" + #"W_All AnalogUpALM" + #"W_All AnalogLowALM" + #"W_All OtherALM";
END_REGION

REGION Network 36: 故障累加5
   RUNG wire#powerrail
      Add(in1 := #"W_All SensALM"[1], in2 := #"W_All SensALM"[2], in3 := #"W_All SensALM"[3], in4 := #"W_All SensALM"[4], in5 := #"W_All SensALM"[5], in6 := #"W_All SensALM"[6], in7 := #"W_All MoveALM"[1], in8 := #"W_All MoveALM"[2], in9 := #"W_All MoveALM"[3], out => #WD_RealTimeALM[10])
   END_RUNG
   // the same network as SCL:
   #WD_RealTimeALM[10] := #"W_All SensALM"[1] + #"W_All SensALM"[2] + #"W_All SensALM"[3] + #"W_All SensALM"[4] + #"W_All SensALM"[5] + #"W_All SensALM"[6] + #"W_All MoveALM"[1] + #"W_All MoveALM"[2] + #"W_All MoveALM"[3];
END_REGION

REGION Network 37: 故障累加6
   RUNG wire#powerrail
      Add(in1 := #WD_RealTimeALM[1], in2 := #WD_RealTimeALM[2], in3 := #WD_RealTimeALM[3], in4 := #WD_RealTimeALM[4], in5 := #WD_RealTimeALM[5], in6 := #WD_RealTimeALM[6], in7 := #WD_RealTimeALM[7], in8 := #WD_RealTimeALM[8], in9 := #WD_RealTimeALM[9], in10 := #WD_RealTimeALM[10], out => #WD_RealTimeALM[15])
   END_RUNG
   // the same network as SCL:
   #WD_RealTimeALM[15] := #WD_RealTimeALM[1] + #WD_RealTimeALM[2] + #WD_RealTimeALM[3] + #WD_RealTimeALM[4] + #WD_RealTimeALM[5] + #WD_RealTimeALM[6] + #WD_RealTimeALM[7] + #WD_RealTimeALM[8] + #WD_RealTimeALM[9] + #WD_RealTimeALM[10];
END_REGION

REGION Network 38: 故障数据转存
   RUNG wire#powerrail
      P_Contact(operand := #"M_All ALM", bit := #M_Pluse[1])
      wire#w1
      { S7_Templates := "SrcType := DInt" } GT_Contact(in1 := #WD_RealTimeALM[15], in2 := 0)
      Move(in := #WD_RealTimeALM[15], out1 => #WD_OldTimeALM[1])
   END_RUNG
   RUNG wire#powerrail
      P_Contact(operand := #MT_ErrTime[1].Q, bit := #M_Pluse[2])
   END_RUNG wire#w1
   // the same network as SCL:
   #_w1 := #"M_All ALM" AND NOT #M_Pluse[1];   // rising edge of #"M_All ALM"
   #M_Pluse[1] := #"M_All ALM";
   #_w2 := #MT_ErrTime[1].Q AND NOT #M_Pluse[2];   // rising edge of #MT_ErrTime[1].Q
   #M_Pluse[2] := #MT_ErrTime[1].Q;
   IF (#_w1 OR #_w2) AND (#WD_RealTimeALM[15] > 0) THEN #WD_OldTimeALM[1] := #WD_RealTimeALM[15]; END_IF;
END_REGION

REGION Network 39: 故障汇总新的
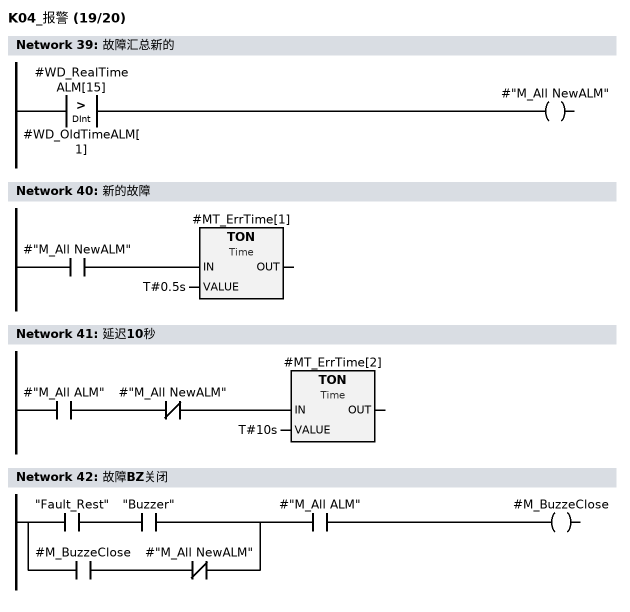
   RUNG wire#powerrail
      { S7_Templates := "SrcType := DInt" } GT_Contact(in1 := #WD_RealTimeALM[15], in2 := #WD_OldTimeALM[1])
      Coil( #"M_All NewALM" )
   END_RUNG
   // the same network as SCL:
   #"M_All NewALM" := #WD_RealTimeALM[15] > #WD_OldTimeALM[1];
END_REGION

REGION Network 40: 新的故障
   #MT_ErrTime[1].TON(IN := #"M_All NewALM", PT := T#0.5s);   // TON coil
END_REGION

REGION Network 41: 延迟10秒
   #MT_ErrTime[2].TON(IN := #"M_All ALM" AND NOT #"M_All NewALM", PT := T#10s);   // TON coil
END_REGION

REGION Network 42: 故障BZ关闭
   RUNG wire#powerrail
      Contact( "Fault_Rest" )
      Contact( "Buzzer" )
      wire#w1
      Contact( #"M_All ALM" )
      Coil( #M_BuzzeClose )
   END_RUNG
   RUNG wire#powerrail
      Contact( #M_BuzzeClose )
      I_Contact( #"M_All NewALM" )
   END_RUNG wire#w1
   // the same network as SCL:
   #M_BuzzeClose := (("Fault_Rest" AND "Buzzer") OR (#M_BuzzeClose AND NOT #"M_All NewALM")) AND #"M_All ALM";
END_REGION

REGION Network 43: 蜂鸣器
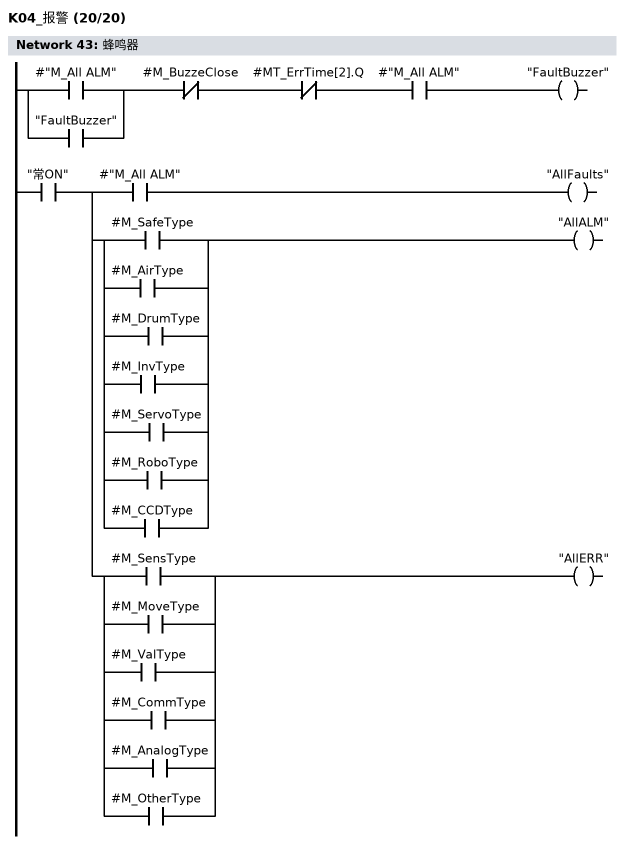
   RUNG wire#powerrail
      Contact( #"M_All ALM" )
      wire#w1
      I_Contact( #M_BuzzeClose )
      I_Contact( #MT_ErrTime[2].Q )
      Contact( #"M_All ALM" )
      Coil( "FaultBuzzer" )
   END_RUNG
   RUNG wire#powerrail
      Contact( "FaultBuzzer" )
   END_RUNG wire#w1
   RUNG wire#powerrail
      Contact( "常ON" )
      wire#w2
      Contact( #"M_All ALM" )
      Coil( "AllFaults" )
   END_RUNG
   RUNG wire#w2
      Contact( #M_SafeType )
      wire#w3
      Coil( "AllALM" )
   END_RUNG
   RUNG wire#w2
      Contact( #M_AirType )
   END_RUNG wire#w3
   RUNG wire#w2
      Contact( #M_DrumType )
   END_RUNG wire#w3
   RUNG wire#w2
      Contact( #M_InvType )
   END_RUNG wire#w3
   RUNG wire#w2
      Contact( #M_ServoType )
   END_RUNG wire#w3
   RUNG wire#w2
      Contact( #M_RoboType )
   END_RUNG wire#w3
   RUNG wire#w2
      Contact( #M_CCDType )
   END_RUNG wire#w3
   RUNG wire#w2
      Contact( #M_SensType )
      wire#w4
      Coil( "AllERR" )
   END_RUNG
   RUNG wire#w2
      Contact( #M_MoveType )
   END_RUNG wire#w4
   RUNG wire#w2
      Contact( #M_ValType )
   END_RUNG wire#w4
   RUNG wire#w2
      Contact( #M_CommType )
   END_RUNG wire#w4
   RUNG wire#w2
      Contact( #M_AnalogType )
   END_RUNG wire#w4
   RUNG wire#w2
      Contact( #M_OtherType )
   END_RUNG wire#w4
   // the same network as SCL:
   "FaultBuzzer" := (#"M_All ALM" OR "FaultBuzzer") AND NOT #M_BuzzeClose AND NOT #MT_ErrTime[2].Q AND #"M_All ALM";
   "AllFaults" := "常ON" AND #"M_All ALM";
   "AllALM" := "常ON" AND (#M_SafeType OR #M_AirType OR #M_DrumType OR #M_InvType OR #M_ServoType OR #M_RoboType OR #M_CCDType);
   "AllERR" := "常ON" AND (#M_SensType OR #M_MoveType OR #M_ValType OR #M_CommType OR #M_AnalogType OR #M_OtherType);
END_REGION
END_FUNCTION_BLOCK
